% RSLogix 500 project Automatisierte Nussfüllstation.RSS, saved by version 8.30.00.16 %
PROJECT "UNTITLED"    % processor: Bul.1763 MicroLogix 1100 Series B %

PROGRAM FILES
  LAD 2 "MAIN"  3 rungs
  LAD 3 "DIGITAL IO"  8 rungs
  LAD 4 "CONTROLS"  6 rungs

DATA FILES
  O0 OUTPUT  4 elements
  I1 INPUT  6 elements
  S2 STATUS  66 elements
  B3 BINARY  2 elements
  T4 TIMER  5 elements
  C5 COUNTER  1 elements
  R6 CONTROL  1 elements
  N7 INTEGER  1 elements
  F8 FLOAT  1 elements

LADDER 2 "MAIN"
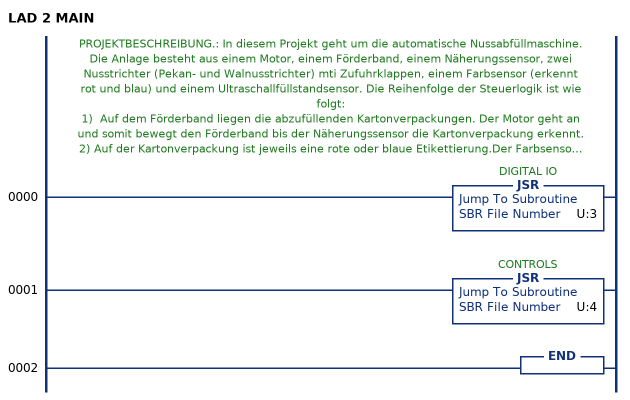
% Rung: 0 %
% PROJEKTBESCHREIBUNG.: In diesem Projekt geht um die automatische Nussabfüllmaschine. Die Anlage besteht aus einem Motor, einem Förderband, einem Näherungssensor, zwei Nusstrichter (Pekan- und Walnusstrichter) mti Zufuhrklappen, einem Farbsensor (erkennt rot und blau) und einem Ultraschallfüllstandsensor. Die Reihenfolge der Steuerlogik ist wie folgt:
% 1)  Auf dem Förderband liegen die abzufüllenden Kartonverpackungen. Der Motor geht an und somit bewegt den Förderband bis der Näherungssensor die Kartonverpackung erkennt.
% 2) Auf der Kartonverpackung ist jeweils eine rote oder blaue Etikettierung.Der Farbsensor erkennt die Farbe und anhand dieser Farbe (rot für Pekannüsse und blau für Walnüsse) wird jeweiligen Zufuhrklappen zur Befüllung geöffnet.
% 3) Der Ultraschallfüllstandsensor misst ständig ,ob die Verpackung voll ist. Falls ja, die Zufuhrklappe ist geschlossen und der Förderband bewegt die befüllte Verpackung weiter. %
SOR JSR U:3 EOR
%   U:3  "DIGITAL IO" %
% Rung: 1 %
SOR JSR U:4 EOR
%   U:4  "CONTROLS" %
% Rung: 2 %
SOR END EOR

LADDER 3 "DIGITAL IO"
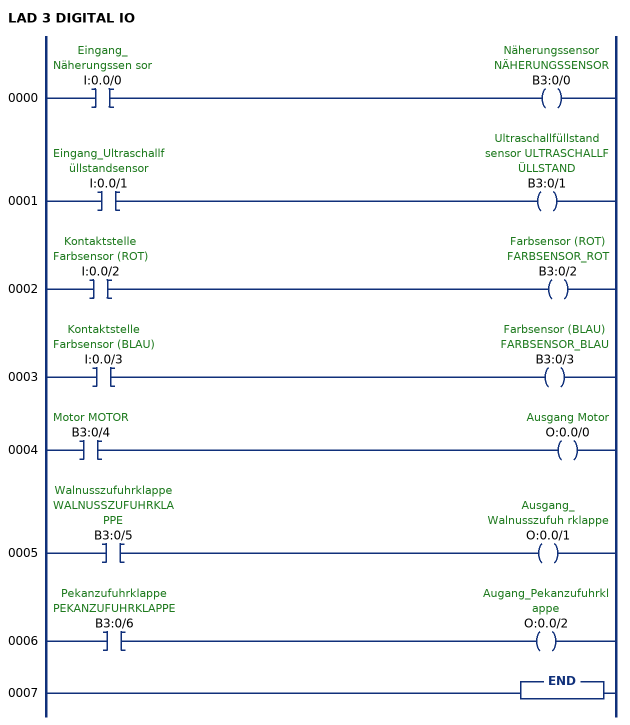
% Rung: 0 %
SOR XIC I:0.0/0 OTE B3:0/0 EOR
%   I:0.0/0  "Eingang_Näherungssen sor" %
%   B3:0/0  NÄHERUNGSSENSOR  "Näherungssensor" %
% Rung: 1 %
SOR XIC I:0.0/1 OTE B3:0/1 EOR
%   I:0.0/1  "Eingang_Ultraschallf üllstandsensor" %
%   B3:0/1  ULTRASCHALLFÜLLSTAND  "Ultraschallfüllstand sensor" %
% Rung: 2 %
SOR XIC I:0.0/2 OTE B3:0/2 EOR
%   I:0.0/2  "Kontaktstelle Farbsensor (ROT)" %
%   B3:0/2  FARBSENSOR_ROT  "Farbsensor (ROT)" %
% Rung: 3 %
SOR XIC I:0.0/3 OTE B3:0/3 EOR
%   I:0.0/3  "Kontaktstelle Farbsensor (BLAU)" %
%   B3:0/3  FARBSENSOR_BLAU  "Farbsensor (BLAU)" %
% Rung: 4 %
SOR XIC B3:0/4 OTE O:0.0/0 EOR
%   B3:0/4  MOTOR  "Motor" %
%   O:0.0/0  "Ausgang Motor" %
% Rung: 5 %
SOR XIC B3:0/5 OTE O:0.0/1 EOR
%   B3:0/5  WALNUSSZUFUHRKLAPPE  "Walnusszufuhrklappe" %
%   O:0.0/1  "Ausgang_Walnusszufuh rklappe" %
% Rung: 6 %
SOR XIC B3:0/6 OTE O:0.0/2 EOR
%   B3:0/6  PEKANZUFUHRKLAPPE  "Pekanzufuhrklappe" %
%   O:0.0/2  "Augang_Pekanzufuhrkl appe" %
% Rung: 7 %
SOR END EOR

LADDER 4 "CONTROLS"
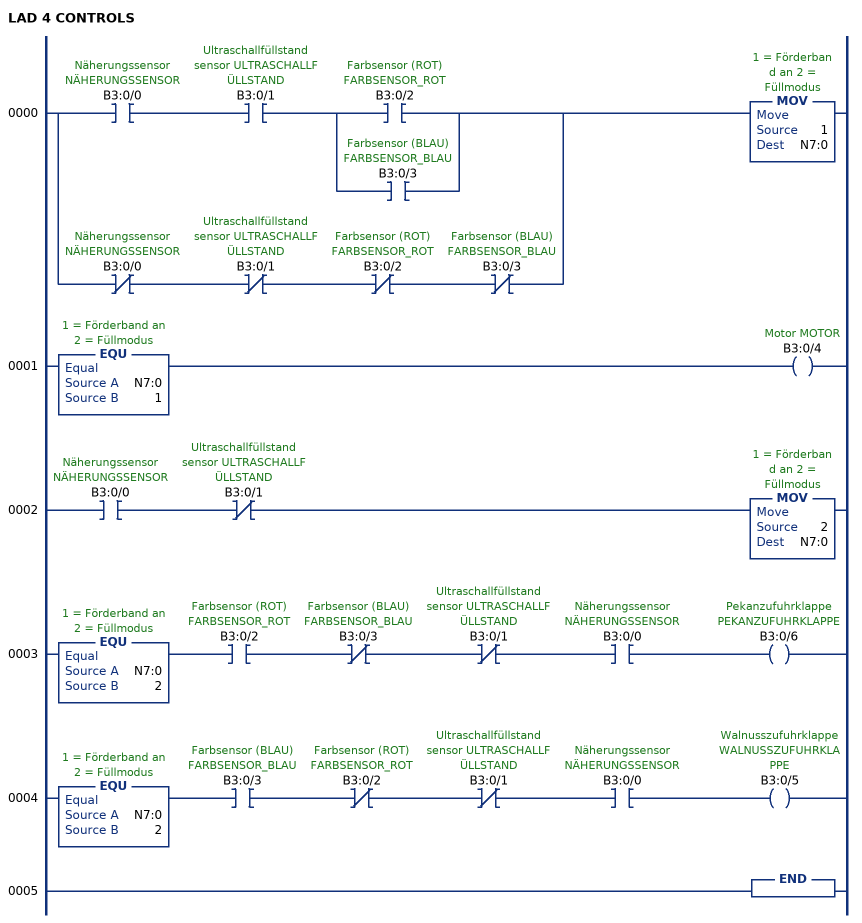
% Rung: 0 %
SOR BST XIC B3:0/0 XIC B3:0/1 BST XIC B3:0/2 NXB XIC B3:0/3 BND NXB XIO B3:0/0 XIO B3:0/1 XIO B3:0/2 XIO B3:0/3 BND MOV 1 N7:0 EOR
%   B3:0/0  NÄHERUNGSSENSOR  "Näherungssensor" %
%   B3:0/1  ULTRASCHALLFÜLLSTAND  "Ultraschallfüllstand sensor" %
%   B3:0/2  FARBSENSOR_ROT  "Farbsensor (ROT)" %
%   B3:0/3  FARBSENSOR_BLAU  "Farbsensor (BLAU)" %
%   N7:0  "1 = Förderband an 2 = Füllmodus" %
% Rung: 1 %
SOR EQU N7:0 1 OTE B3:0/4 EOR
%   N7:0  "1 = Förderband an 2 = Füllmodus" %
%   B3:0/4  MOTOR  "Motor" %
% Rung: 2 %
SOR XIC B3:0/0 XIO B3:0/1 MOV 2 N7:0 EOR
%   B3:0/0  NÄHERUNGSSENSOR  "Näherungssensor" %
%   B3:0/1  ULTRASCHALLFÜLLSTAND  "Ultraschallfüllstand sensor" %
%   N7:0  "1 = Förderband an 2 = Füllmodus" %
% Rung: 3 %
SOR EQU N7:0 2 XIC B3:0/2 XIO B3:0/3 XIO B3:0/1 XIC B3:0/0 OTE B3:0/6 EOR
%   N7:0  "1 = Förderband an 2 = Füllmodus" %
%   B3:0/2  FARBSENSOR_ROT  "Farbsensor (ROT)" %
%   B3:0/3  FARBSENSOR_BLAU  "Farbsensor (BLAU)" %
%   B3:0/1  ULTRASCHALLFÜLLSTAND  "Ultraschallfüllstand sensor" %
%   B3:0/0  NÄHERUNGSSENSOR  "Näherungssensor" %
%   B3:0/6  PEKANZUFUHRKLAPPE  "Pekanzufuhrklappe" %
% Rung: 4 %
SOR EQU N7:0 2 XIC B3:0/3 XIO B3:0/2 XIO B3:0/1 XIC B3:0/0 OTE B3:0/5 EOR
%   N7:0  "1 = Förderband an 2 = Füllmodus" %
%   B3:0/3  FARBSENSOR_BLAU  "Farbsensor (BLAU)" %
%   B3:0/2  FARBSENSOR_ROT  "Farbsensor (ROT)" %
%   B3:0/1  ULTRASCHALLFÜLLSTAND  "Ultraschallfüllstand sensor" %
%   B3:0/0  NÄHERUNGSSENSOR  "Näherungssensor" %
%   B3:0/5  WALNUSSZUFUHRKLAPPE  "Walnusszufuhrklappe" %
% Rung: 5 %
SOR END EOR

OTHER DOCUMENTED ADDRESSES
  B3:0/7  "Motorstart-bit"
  B3:0/8  "ONS"
  B3:0/9  "Motor-Trigger"
  B3:0/10  "ONS"
  B3:0/11  "Motor-Interrupt"
  B3:0/12  "Walnusszufuhrklappe- trigger"
  B3:0/13  "ONS"
  B3:0/14  "Befüllvorgang- interrupt"
  B3:0/15  "ONS"
  B3:1/0  "Pekanzufuhrklappe- trigger"
  B3:1/1  "Motorstart-Bit"
  T4:0  "Motoreinschaltverzög erung"
  T4:1  "Motorausschaltverzög erung"
  T4:2  "Walnusstrichterverzö gerung"
  T4:3  "Befüllvorgang- Interrupt- Verzögerung"
  T4:4  "Pekanzufuhrklappever zögerung"

COMMENTS NOT ATTACHED TO A CURRENT RUNG
  T4:0: Die Logikpfaden 1-4 enthalten die Steuerlogik für Motor
  T4:2: Die Logikpfade 5-12 enthalten Steuerlogik zur Befüllen von Leere Kisten anhand der Etikettfarbe

DATA TABLE (non-zero values as saved)
DATA B3
% B3:0 % 0X0180 0X0000
DATA T4
% .PRE .ACC %
% T4:0 % 10 10
% T4:1 % 10 0
% T4:2 % 10 0
% T4:3 % 10 0
% T4:4 % 10 0
